{attribute 'qualified_only'}
{attribute 'to_string'}
TYPE E_POS :			// Position numbers
(
	UNDEFINED := 0,
	
	// Special case for alarm handler	
	ACCEPT_ANY := 1,

	MAIN :=		10,
	

	
	
	MUST_BE_LAST	// ALWAYS KEEP THIS LAST!!!
);
END_TYPE

(* stored: Version 1.1.0.1, ProductVersion 3.1.4026.18
   DUT E_POS: Id {0993ecb2-dd65-03af-3a68-026bf576fae3} *)
